KUKA KRL data list: style_1.dat

&ACCESS RVO1
&REL 101
&COMMENT GE4_002
DEFDAT  style_1
;FOLD EXTERNAL DECLARATIONS;%{PE}%MKUKATPBASIS,%CEXT,%VCOMMON,%P
;FOLD BASISTECH EXT;%{PE}%MKUKATPBASIS,%CEXT,%VEXT,%P
EXT  BAS (BAS_COMMAND  :IN,REAL  :IN )
DECL INT SUCCESS
;ENDFOLD (BASISTECH EXT)
;FOLD USER EXT;%{E}%MKUKATPUSER,%CEXT,%VEXT,%P
;Make your modifications here

;ENDFOLD (USER EXT)
;ENDFOLD (EXTERNAL DECLARATIONS)
DECL BASIS_SUGG_T LAST_BASIS={POINT1[] "POUNCE                  ",POINT2[] "POUNCE                  ",CP_PARAMS[] "CPDAT0                  ",PTP_PARAMS[] "PDAT6                   ",CONT[] "                        ",CP_VEL[] "2.0                     ",PTP_VEL[] "90                      ",SYNC_PARAMS[] "SYNCDAT                 ",SPL_NAME[] "S0                      ",A_PARAMS[] "ADAT0                   "}
ENDDAT
